Staubli VAL3: CMS_Module.pjx

--- CMS_Module.pjx ---
Parameters version=s8.10.2Cs9_BS1991 stackSize=20000 millimeterUnit=true
Program file=clkAirexOff.pgx
Program file=clkAirexOn.pgx
Program file=clkAllOff.pgx
Program file=clkAllOn.pgx
Program file=clkBack.pgx
Program file=clkCleanupChuck1.pgx
Program file=clkCleanupChuck2.pgx
Program file=clkDoAirex.pgx
Program file=clkDoModules.pgx
Program file=clkGlueGlass.pgx
Program file=clkPark1.pgx
Program file=clkPark2.pgx
Program file=clkValve0.pgx
Program file=clkValve1.pgx
Program file=clkValve10.pgx
Program file=clkValve11.pgx
Program file=clkValve12.pgx
Program file=clkValve13.pgx
Program file=clkValve14.pgx
Program file=clkValve15.pgx
Program file=clkValve16.pgx
Program file=clkValve17.pgx
Program file=clkValve2.pgx
Program file=clkValve3.pgx
Program file=clkValve4.pgx
Program file=clkValve5.pgx
Program file=clkValve6.pgx
Program file=clkValve7.pgx
Program file=clkValve8.pgx
Program file=clkValve9.pgx
Program file=clkValvePage.pgx
Program file=doAirex.pgx
Program file=doModules.pgx
Program file=glueGlass.pgx
Program file=goRemote.pgx
Program file=moveDown.pgx
Program file=moveStampUp.pgx
Program file=park1.pgx
Program file=print.pgx
Program file=selectedCheck.pgx
Program file=selectedClear.pgx
Program file=setSpeed.pgx
Program file=setValveStatus.pgx
Program file=socketServer.pgx
Program file=start.pgx
Program file=stop.pgx
Program file=toggleValve.pgx
Data file=CMS_Module.dtx

--- CMS_Module.dtx ---
bool bDoAirex = true
bool bGlueGlass
public dio doJ206_EtherCAT_Box_1__CPX_FB37__Q0 = {link=J206_EtherCAT\Box_1_(CPX-FB37)\%Q0}
public dio doJ206_EtherCAT_Box_1__CPX_FB37__Q1 = {link=J206_EtherCAT\Box_1_(CPX-FB37)\%Q1}
public dio doJ206_EtherCAT_Box_1__CPX_FB37__Q10 = {link=J206_EtherCAT\Box_1_(CPX-FB37)\%Q10}
public dio doJ206_EtherCAT_Box_1__CPX_FB37__Q11 = {link=J206_EtherCAT\Box_1_(CPX-FB37)\%Q11}
public dio doJ206_EtherCAT_Box_1__CPX_FB37__Q12 = {link=J206_EtherCAT\Box_1_(CPX-FB37)\%Q12}
public dio doJ206_EtherCAT_Box_1__CPX_FB37__Q13 = {link=J206_EtherCAT\Box_1_(CPX-FB37)\%Q13}
public dio doJ206_EtherCAT_Box_1__CPX_FB37__Q14 = {link=J206_EtherCAT\Box_1_(CPX-FB37)\%Q14}
public dio doJ206_EtherCAT_Box_1__CPX_FB37__Q15 = {link=J206_EtherCAT\Box_1_(CPX-FB37)\%Q15}
public dio doJ206_EtherCAT_Box_1__CPX_FB37__Q16 = {link=J206_EtherCAT\Box_1_(CPX-FB37)\%Q16}
public dio doJ206_EtherCAT_Box_1__CPX_FB37__Q17 = {link=J206_EtherCAT\Box_1_(CPX-FB37)\%Q17}
public dio doJ206_EtherCAT_Box_1__CPX_FB37__Q18 = {link=J206_EtherCAT\Box_1_(CPX-FB37)\%Q18}
public dio doJ206_EtherCAT_Box_1__CPX_FB37__Q19 = {link=J206_EtherCAT\Box_1_(CPX-FB37)\%Q19}
public dio doJ206_EtherCAT_Box_1__CPX_FB37__Q2 = {link=J206_EtherCAT\Box_1_(CPX-FB37)\%Q2}
public dio doJ206_EtherCAT_Box_1__CPX_FB37__Q20 = {link=J206_EtherCAT\Box_1_(CPX-FB37)\%Q20}
public dio doJ206_EtherCAT_Box_1__CPX_FB37__Q21 = {link=J206_EtherCAT\Box_1_(CPX-FB37)\%Q21}
public dio doJ206_EtherCAT_Box_1__CPX_FB37__Q22 = {link=J206_EtherCAT\Box_1_(CPX-FB37)\%Q22}
public dio doJ206_EtherCAT_Box_1__CPX_FB37__Q23 = {link=J206_EtherCAT\Box_1_(CPX-FB37)\%Q23}
public dio doJ206_EtherCAT_Box_1__CPX_FB37__Q24 = {link=J206_EtherCAT\Box_1_(CPX-FB37)\%Q24}
public dio doJ206_EtherCAT_Box_1__CPX_FB37__Q25 = {link=J206_EtherCAT\Box_1_(CPX-FB37)\%Q25}
public dio doJ206_EtherCAT_Box_1__CPX_FB37__Q26 = {link=J206_EtherCAT\Box_1_(CPX-FB37)\%Q26}
public dio doJ206_EtherCAT_Box_1__CPX_FB37__Q27 = {link=J206_EtherCAT\Box_1_(CPX-FB37)\%Q27}
public dio doJ206_EtherCAT_Box_1__CPX_FB37__Q28 = {link=J206_EtherCAT\Box_1_(CPX-FB37)\%Q28}
public dio doJ206_EtherCAT_Box_1__CPX_FB37__Q29 = {link=J206_EtherCAT\Box_1_(CPX-FB37)\%Q29}
public dio doJ206_EtherCAT_Box_1__CPX_FB37__Q3 = {link=J206_EtherCAT\Box_1_(CPX-FB37)\%Q3}
public dio doJ206_EtherCAT_Box_1__CPX_FB37__Q30 = {link=J206_EtherCAT\Box_1_(CPX-FB37)\%Q30}
public dio doJ206_EtherCAT_Box_1__CPX_FB37__Q31 = {link=J206_EtherCAT\Box_1_(CPX-FB37)\%Q31}
public dio doJ206_EtherCAT_Box_1__CPX_FB37__Q4 = {link=J206_EtherCAT\Box_1_(CPX-FB37)\%Q4}
public dio doJ206_EtherCAT_Box_1__CPX_FB37__Q5 = {link=J206_EtherCAT\Box_1_(CPX-FB37)\%Q5}
public dio doJ206_EtherCAT_Box_1__CPX_FB37__Q6 = {link=J206_EtherCAT\Box_1_(CPX-FB37)\%Q6}
public dio doJ206_EtherCAT_Box_1__CPX_FB37__Q7 = {link=J206_EtherCAT\Box_1_(CPX-FB37)\%Q7}
public dio doJ206_EtherCAT_Box_1__CPX_FB37__Q8 = {link=J206_EtherCAT\Box_1_(CPX-FB37)\%Q8}
public dio doJ206_EtherCAT_Box_1__CPX_FB37__Q9 = {link=J206_EtherCAT\Box_1_(CPX-FB37)\%Q9}
public dio switchMagnet = {link=FastIO\fOut0}
public dio switchVac0 = {link=ValveIO\valve1}
public dio switchVac1 = {link=ValveIO\valve2}
frame fPalette = {x=-254.28, y=175.62, z=30, rz=0.110016, fatherId=world[0]}
jointRs jInitialPosition = {j1=50, j2=50, j3=80, j4=15}
jointRs jRestPosition = {j1=70, j2=40, j3=80, j4=10}
mdesc mFast = {accel=20, vel=50, decel=20, leave=100}
mdesc mNomSpeed = {accel=10, vel=30, decel=10}
mdesc mSlow = {accel=5, vel=20, decel=5, tmax=99, rmax=99, leave=25, reach=25}
num airexValve[6]
  [0] = 12
  [1] = 6
  [3] = 13
  [4] = 7
  [5] = 1
num hdiValve[6]
  [0] = 14
  [1] = 8
  [2] = 2
  [3] = 16
  [4] = 10
  [5] = 4
num nError
num sensorValve[6]
  [0] = 15
  [1] = 9
  [2] = 3
  [3] = 17
  [4] = 11
  [5] = 5
num statusValves[32]
  [0] = 1
  [1] = 1
  [2] = 1
  [3] = 1
  [4] = 1
  [5] = 1
  [6] = 1
  [7] = 1
  [8] = 1
  [9] = 1
  [10] = 1
  [11] = 1
  [12] = 1
  [13] = 1
  [14] = 1
  [15] = 1
  [16] = 1
  [17] = 1
  [18] = 1
  [19] = 1
  [20] = 1
  [21] = 1
  [22] = 1
  [23] = 1
  [24] = 1
  [25] = 1
  [26] = 1
  [27] = 1
  [28] = 1
  [29] = 1
  [30] = 1
  [31] = 1
num waitGlue = 3
num waitShort = 1
pointRs airexFinal[6]
  [0] = {x=59, y=184, z=-97.69, rx=180, fatherId=fPalette[0]}
  [1] = {x=134, y=184, z=-97.69, rx=180, fatherId=fPalette[0]}
  [2] = {x=209, y=184, z=-97.69, rx=180, fatherId=fPalette[0]}
  [3] = {x=59, y=314, z=-97.69, rx=180, fatherId=fPalette[0]}
  [4] = {x=134, y=314, z=-97.69, rx=180, fatherId=fPalette[0]}
  [5] = {x=209, y=314, z=-97.69, rx=180, fatherId=fPalette[0]}
pointRs airexGlueStampEnd = {x=466.48, y=113.596594, z=-96.5, rx=180, ry=6.951996E-15, rz=0.0536958, fatherId=fPalette[0]}
pointRs airexGlueStampHome = {x=496, y=54, z=-97.69, rx=180, fatherId=fPalette[0]}
pointRs airexInitial[6]
  [0] = {x=59, y=113.6, z=-97.69, rx=180, fatherId=fPalette[0]}
  [1] = {x=134, y=113.6, z=-97.69, rx=180, fatherId=fPalette[0]}
  [2] = {x=209, y=113.6, z=-97.69, rx=180, fatherId=fPalette[0]}
  [3] = {x=59, y=144, z=-97.69, rx=180, fatherId=fPalette[0]}
  [4] = {x=134, y=144, z=-97.69, rx=180, fatherId=fPalette[0]}
  [5] = {x=209, y=144, z=-97.69, rx=180, fatherId=fPalette[0]}
pointRs chuck1[6]
  [0] = {x=59, y=39, z=-97.69, rx=180, fatherId=fPalette[0]}
  [1] = {x=134, y=39, z=-97.69, rx=180, fatherId=fPalette[0]}
  [2] = {x=209, y=39, z=-97.69, rx=180, fatherId=fPalette[0]}
  [3] = {x=59, y=79, z=-97.69, rx=180, fatherId=fPalette[0]}
  [4] = {x=134, y=79, z=-97.69, rx=180, fatherId=fPalette[0]}
  [5] = {x=209, y=79, z=-97.69, rx=180, fatherId=fPalette[0]}
pointRs chuck2[6]
  [0] = {x=291, y=54, z=-97.69, rx=180, fatherId=fPalette[0]}
  [1] = {x=361, y=54, z=-97.69, rx=180, fatherId=fPalette[0]}
  [2] = {x=291, y=119, z=-97.69, rx=180, fatherId=fPalette[0]}
  [3] = {x=361, y=119, z=-97.69, rx=180, fatherId=fPalette[0]}
  [4] = {x=291, y=184, z=-97.69, rx=180, fatherId=fPalette[0]}
  [5] = {x=361, y=184, z=-97.69, rx=180, fatherId=fPalette[0]}
pointRs gluePickPoint[6]
  [0] = {x=260, y=-15.8, z=-62.5, rx=180, ry=6.952208E-15, rz=0.0408868, fatherId=world[0]}
  [1] = {x=260, y=17.2, z=-62.5, rx=180, fatherId=world[0]}
  [2] = {x=290, y=-15.8, z=-62.5, rx=180, fatherId=world[0]}
  [3] = {x=290, y=17.2, z=-62.5, rx=180, fatherId=world[0]}
  [4] = {x=320, y=-15.8, z=-62.5, rx=180, fatherId=world[0]}
  [5] = {x=320, y=17.2, z=-62.5, rx=180, fatherId=world[0]}
pointRs hdiFinal[6]
  [0] = {x=59, y=249, z=-97.69, rx=180, fatherId=fPalette[0]}
  [1] = {x=134, y=249, z=-97.69, rx=180, fatherId=fPalette[0]}
  [2] = {x=209, y=249, z=-97.69, rx=180, fatherId=fPalette[0]}
  [3] = {x=59, y=379, z=-97.69, rx=180, fatherId=fPalette[0]}
  [4] = {x=134, y=379, z=-97.69, rx=180, fatherId=fPalette[0]}
  [5] = {x=209, y=379, z=-97.69, rx=180, fatherId=fPalette[0]}
pointRs pBasisRs = {x=-45.372705, y=215.0412411, z=72.706789, rx=180, ry=6.952541E-15, rz=0.0207374, fatherId=world[0]}
pointRs pFrameUrsprung = {x=-254.28, y=175.62, z=30, fatherId=world[0]}
pointRs pFrameX = {x=271.72, y=176.63, z=30, fatherId=world[0]}
pointRs pFrameY = {x=-255.12, y=613.62, z=30, fatherId=world[0]}
string colorOff = "beige"
string colorOn = "darkgreen"
string colorValveButton[32]
  [0] = "darkgreen"
  [1] = "darkgreen"
  [2] = "darkgreen"
  [3] = "darkgreen"
  [4] = "darkgreen"
  [5] = "darkgreen"
  [6] = "darkgreen"
  [7] = "darkgreen"
  [8] = "darkgreen"
  [9] = "darkgreen"
  [10] = "darkgreen"
  [11] = "darkgreen"
  [12] = "darkgreen"
  [13] = "darkgreen"
  [14] = "darkgreen"
  [15] = "darkgreen"
  [16] = "darkgreen"
  [17] = "darkgreen"
  [18] = "darkgreen"
  [19] = "darkgreen"
  [20] = "darkgreen"
  [21] = "darkgreen"
  [22] = "darkgreen"
  [23] = "darkgreen"
  [24] = "darkgreen"
  [25] = "darkgreen"
  [26] = "darkgreen"
  [27] = "darkgreen"
  [28] = "darkgreen"
  [29] = "darkgreen"
  [30] = "darkgreen"
  [31] = "darkgreen"
public tool tTool = {z=70, rz=-97.72, fatherId=flange[0]}
trsf trApproach = {z=-20}
trsf trStamp = {z=-6}
trsf trZsafe = {z=-70}
string colorVacuumStatus1
string statusDoAirex
string colorGray
string colorRunning
string colorCleanupChuck1
string statusCleanupChuck1
mdesc mVerySlow = {accel=2, vel=5, decel=2, tmax=5, rmax=5, leave=10, reach=10}
string statusDoModules
string statusCleanupChuck2
string colorCleanupChuck2
bool bDoModules
pointRs gluePickPoint2[6]
  [0] = {x=360, y=-25, z=-62.5, rx=180, ry=6.952208E-15, rz=0.0408868, fatherId=world[0]}
  [1] = {x=360, y=25, z=-62.5, rx=180, fatherId=world[0]}
  [2] = {x=410, y=-25, z=-62.5, rx=180, fatherId=world[0]}
  [3] = {x=410, y=25, z=-62.5, rx=180, fatherId=world[0]}
  [4] = {x=460, y=-25, z=-62.5, rx=180, fatherId=world[0]}
  [5] = {x=460, y=25, z=-62.5, rx=180, fatherId=world[0]}
pointRs moduleGlueStampHome = {x=436, y=54, z=-97.69, rx=180, ry=6.951996E-15, fatherId=fPalette[0]}
pointRs moduleGlueStampEnd = {x=466.48, y=156.596594, z=-96.5, rx=180, ry=6.951996E-15, rz=0.0536958, fatherId=fPalette[0]}
mdesc mExtremelySlow = {accel=0.05, vel=0.05, decel=0.05, tmax=0.04, rmax=0.04, leave=1, reach=1}
pointRs glueFirstPoint[2]
  [0] = {x=350, y=-15.8, z=-62.5, rx=180, ry=6.952208E-15, rz=0.0408868, fatherId=world[0]}
  [1] = {x=310, y=-25, z=-62.5, rx=180, rz=0.0408868, fatherId=world[0]}
trsf trZclose = {z=-10}
bool bSelectItem
bool bSelectedItems[6]
bool bSkipGlue
string colorError
string strStatus
trsf trZero
pointRs pSomewhere = {x=300, y=200, fatherId=world[0]}
trsf trPressTwo = {z=2}
trsf trUpTwo = {z=-8}
jointRs jPosition
string sPosition
bool bCleanup
num speedFactor
mdesc mSpeedArray[10]
  [0] = {accel=0.05, vel=0.05, decel=0.05, tmax=0.04, rmax=0.04, leave=1, reach=1}
  [1] = {accel=0.5, vel=0.5, decel=0.5, tmax=1, rmax=1, leave=2, reach=2}
  [2] = {accel=1, vel=1, decel=1, tmax=2, rmax=2, leave=2, reach=2}
  [3] = {accel=2, vel=2, decel=2, tmax=5, rmax=5, leave=5, reach=5}
  [4] = {accel=4, vel=5, decel=4, tmax=10, rmax=10, leave=10, reach=10}
  [5] = {accel=5, vel=7, decel=5, tmax=15, rmax=15, leave=20, reach=10}
  [6] = {accel=6, vel=10, decel=6, tmax=20, rmax=20, leave=20, reach=10}
  [7] = {accel=8, vel=15, decel=8, tmax=30, rmax=30, leave=40, reach=20}
  [8] = {accel=10, vel=20, decel=10, tmax=60, rmax=60, leave=40, reach=20}
  [9] = {accel=15, vel=30, decel=15, tmax=60, rmax=60, leave=80, reach=40}
trsf trDownTwo = {z=-2}
trsf trUpThree = {z=-9}
trsf trZverySafe = {z=-80}
string version
public sio sioSockets_server = {link=Socket\server}
string sReceiveMsg
string sSendMsg
public sio sioSockets_client = {link=Socket\client}
bool bGoRemote
string strTCPIP
bool bSockets
pointRs pGoRemoteTarget = {fatherId=fPalette[0]}

--- start.pgx ---
program start()
  local num nIndex
begin

  call print("Welcome to TEPX module production")
  version = "2024/12/20-07"

  strTCPIP = "TCP/IP sockets not activated"
  bSockets = false

  // -- required for local automatic?
  if esStatus() == 1
    setSafetyRestart()
  endIf
  if workingMode()==3
    if isPowered() == false
      enablePower()
    endIf
  endIf

  // -- define colors for valve buttons
  colorOff     = "beige"
  colorOn      = "darkgreen"
  colorGray    = "gray"
  colorRunning = "yellow"
  colorError   = "red"

  // -- initialize valve buttons and status
  call setValveStatus()
  for nIndex = 0 to 31
    if statusValves[nIndex] == 0
      colorValveButton[nIndex] = colorOff
    else
      colorValveButton[nIndex] = colorOn
    endIf
  endFor

  // -- initialize selection to be all on and bSelectItem to be off
  for nIndex = 0 to 5
    bSelectedItems[nIndex] = true
  endFor
  bSelectItem = false

  // -- initialize
  switchMagnet = false
  switchVac0   = false
  switchVac1   = false
  bDoAirex     = false
  bGlueGlass   = false
  bEndProgram  = false

  // -- airex valve indices
  airexValve[0]=12
  airexValve[1]=6
  airexValve[2]=0
  airexValve[3]=13
  airexValve[4]=7
  airexValve[5]=1

  // -- hdi valve indices
  hdiValve[0]=14
  hdiValve[1]=8
  hdiValve[2]=2
  hdiValve[3]=16
  hdiValve[4]=10
  hdiValve[5]=4

  // -- sensor valve indices
  sensorValve[0]=15
  sensorValve[1]=9
  sensorValve[2]=3
  sensorValve[3]=17
  sensorValve[4]=11
  sensorValve[5]=5

  colorVacuumStatus1 = colorOff
  colorCleanupChuck1 = colorOff
  colorCleanupChuck2 = colorOff

  statusDoAirex       = colorGray
  statusCleanupChuck1 = colorGray
  statusDoModules     = colorGray
  statusCleanupChuck2 = colorGray

  // -- define manual corrections for final placements
  // trXYCorrectionHDI = trXYZero
  trXYCorrectionHDI = trXYCorrection1

  // -- 4 is the production setting (mExtremelySlow = mSpeedArray[0])
  // -- all the rest have faster mExtremelySlow
  speedFactor = 4
  call setSpeed()

  // -- display user page
  userPage("firstpage")

  // -- this is here that fPalette is defined for manual jogs after program has started
  nError=setFrame(pFrameUrsprung, pFrameX, pFrameY, fPalette)
  resetMotion()
  movej(jInitialPosition, tTool, mNomSpeed)
  waitEndMove()

  taskCreate "doAirexTask", 10, doAirex()
  taskCreate "doModulesTask", 10, doModules()
  taskCreate "doGlueGlass", 10, glueGlass()

  // Note: This is activated only after enabling arm power or move/hold button?!
  taskCreate "socketServerTask", 10, socketServer()


  while true
    jPosition = herej()
    sPosition = toString("6.3", jPosition.j3)
    sMovementID = toString("6.3", getMoveId())
  endWhile

end

--- clkCleanupChuck1.pgx ---
program clkCleanupChuck1()
  local num nAirexIdx
begin
  switchMagnet=false
  statusCleanupChuck1 = colorRunning

  call selectedCheck()
  call print("cleanup (airex) start")

  // -- pick vacuum chuck1's and put them back to their original place
  for nAirexIdx=0 to 5
    if !bSelectItem or (bSelectedItems[nAirexIdx]==true)
      call print("put away chuck " + toString("1.0", nAirexIdx))
      // -- move over final airex position (where the chuck is from gluing) and down
      // -- for edge positions make a curve to avoid hitting side bar
      if nAirexIdx == 0 or nAirexIdx == 3
        movej(appro(airexInitial[1], trZsafe), tTool, mFast)
      endIf

      call moveDown(airexFinal[nAirexIdx], mSlow, trZero, false)

      // -- lift chuck1
      switchMagnet=true
      delay(waitShort)
      movel(appro(airexFinal[nAirexIdx], trZsafe), tTool, mSlow)
      //waitEndMove()

      // -- move over/to initial chuck position
      // -- for edge positions make a curve to avoid hitting side bar
      if nAirexIdx == 0 or nAirexIdx == 3
        movej(appro(airexInitial[1], trZsafe), tTool, mFast)
      endIf
      call moveDown(chuck1[nAirexIdx], mSlow, trZero, false)

      // -- release it
      switchMagnet=false

      // -- move up
      movel(appro(chuck1[nAirexIdx], trZsafe), tTool, mSlow)
    endIf
  endFor

  // -- move back somewhere
  call print("parking robot")
  waitEndMove()
  movej(jInitialPosition, tTool, mFast)
  waitEndMove()
  statusCleanupChuck1 = colorOn
  statusDoAirex = colorGray
  call print("cleanup (airex) done")
  //call selectedClear()

end

--- clkCleanupChuck2.pgx ---
program clkCleanupChuck2()
  local num nIdx
begin
  switchMagnet=false
  statusCleanupChuck2 = colorRunning

  call selectedCheck()
  call print("cleanup (modules) start")

  // -- pick vacuum chuck2's and put them back to their original place
  for nIdx=0 to 5
    if !bSelectItem or (bSelectedItems[nIdx]==true)
      call print("put away chuck " + toString("1.0", nIdx))
      // -- move over final hdi position (where the chuck is from gluing) and down
      // -- for edge positions make a curve to avoid hitting side bar
      if nIdx == 0 or nIdx == 3
        movej(appro(airexInitial[1], trZsafe), tTool, mFast)
      endIf

      // test
      if(nIdx==3)
        trXYCorrectionHDI = trXYZero
      else
        trXYCorrectionHDI = trXYCorrection1
      endIf

      call moveDown(hdiFinal[nIdx], mSlow, trPressTwo, false, trXYCorrectionHDI)

      // -- lift chuck2
      switchMagnet=true
      delay(waitShort)
      movel(appro(hdiFinal[nIdx], trZsafe), tTool, mSlow)
      //waitEndMove()

      // -- move over/to initial chuck position
      // -- for edge positions make a curve to avoid hitting side bar
      if nIdx == 0 or nIdx == 3
        movej(appro(airexInitial[1], trZsafe), tTool, mFast)
      endIf
      call moveDown(chuck2[nIdx], mSlow, trZero, false, trXYZero)

      // -- release it
      switchMagnet=false

      // -- move up
      movel(appro(chuck2[nIdx], trZsafe), tTool, mSlow)
    endIf
  endFor

  // -- move back somewhere
  call print("parking robot")
  waitEndMove()
  movej(jInitialPosition, tTool, mFast)
  waitEndMove()
  call print("cleanup (modules) done")
  statusCleanupChuck2 = colorOn
  statusDoModules = colorGray
  //call selectedClear()

end

--- clkDoTest.pgx ---
program clkDoTest()
begin
  bDoTest=true
end

--- clkPark2.pgx ---
program clkPark2()
begin
  // -- move back to initial position
  resetMotion()
  movej(jInitialPosition,tTool,mNomSpeed)
  waitEndMove()
end

--- clkStop.pgx ---
program clkStop()
begin
  bDoAirex = false
  bDoModules = false
  bCleanup = false
end

--- doAirex.pgx ---
program doAirex()
  local num nAirexIdx
  local bool vacuumCheckDone
begin
  vacuumCheckDone = false
  while true
    call parkEndProgram()

    if bDoAirex==true
      call selectedCheck()
      call print("starting doAirex")
      statusDoAirex = colorRunning

      // -- check that relevant vacuum is active
      if !bSelectItem
        // -- check all
        call print("check vacuum on all")
        delay(waitShort)
        for nAirexIdx = 0 to 5
          // -- check only the sensor valves, not the AIREX frame valves (don't care about those)
          if statusValves[sensorValve[nAirexIdx]] == 0
            bDoAirex = false
            statusDoAirex = colorError
            call print("Error: no vacuum at position " + toString("1.0", nAirexIdx))
          endIf
        endFor
      else
        // -- check only those that are selected
        call print("check vacuum on selection")
        delay(waitShort)
        for nAirexIdx = 0 to 5
          if statusValves[sensorValve[nAirexIdx]] == 0 and (bSelectedItems[nAirexIdx]==true)
            bDoAirex = false
            statusDoAirex = colorError
            call print("Error: no vacuum at position " + toString("1.0", nAirexIdx))
          endIf
        endFor
      endIf
      vacuumCheckDone = true
      if bDoAirex == false
        call print("Fix missing vacuum and try again")
        vacuumCheckDone = false
      endIf

    endIf

    // -- return above does not work. It terminates the task!
    if bDoAirex==true and vacuumCheckDone==true
      call setSpeed()

      if bSkipGlue[0]==false
        call print("picking glue stamp")
        // -- pick glue stamp
        call moveDown(airexGlueStampHome, mSlow, trZero, false, trXYZero)
        waitEndMove()
        movel(appro(airexGlueStampHome, trPressTwo), tTool, mVerySlow)
        waitEndMove()
        delay(waitShort)
        switchMagnet=true
        movel(appro(airexGlueStampHome, trZsafe), tTool, mSlow)

        call parkEndProgram()

        // -- double-dip stamp into glue before starting the normal procedure
        call moveDown(glueFirstPoint[1], mSlow, trZero, false, trXYZero)
        delay(waitGlue)
        call moveStampUp(glueFirstPoint[1], mVerySlow, trXYZero)
        call moveDown(glueFirstPoint[0], mSlow, trZero, false, trXYZero)
        delay(waitGlue)
        call moveStampUp(glueFirstPoint[0], mVerySlow, trXYZero)

        call parkEndProgram()

        // -- apply glue stamp to all positions:
        //    divide approach onto /from glue position into two steps
        //    (1) slowly to trApproach above it
        //    (2) extremely slowly down to/up from glue to trApproach
        for nAirexIdx=0 to 5
          if !bSelectItem or (bSelectedItems[nAirexIdx]==true)
            call setSpeed()
            if bDoAirex==true

              call parkEndProgram()

              call print("getting glue for position " + toString("1.0", nAirexIdx))
              call moveDown(gluePickPoint[nAirexIdx], mSlow, trZero, false, trXYZero)
              delay(waitGlue)

              call moveStampUp(gluePickPoint[nAirexIdx], mVerySlow, trXYZero)

              call parkEndProgram()

              // -- move to where the glue should be applied (the final airex position)
              call print("applying glue to position " + toString("1.0", nAirexIdx))
              call moveDown(airexFinal[nAirexIdx], mSlow, trStamp, false, trXYZero)
              delay(waitGlue)
              call moveStampUp(airexFinal[nAirexIdx], mVerySlow, trXYZero)
            endIf
          endIf
        endFor

        // -- Drop glue stamp
        call setSpeed()
        call print("put away glue stamp")
        call moveDown(airexGlueStampEnd, mSlow, trPressTwo, false, trXYZero)
        waitEndMove()
        switchMagnet = false
        movel(appro(airexGlueStampEnd, trZsafe), tTool, mNomSpeed)
      endIf

      if !bSelectItem
        call print("handling all airex frames")
      else
        call print("handling selected airex frames")
      endIf

      // -- pick weighted vacuum chucks and lift airex frames to HDIs
      for nAirexIdx=0 to 5
        if !bSelectItem or (bSelectedItems[nAirexIdx]==true)
          call setSpeed()
          if bDoAirex==true
            // -- move over/to chuck
            call moveDown(chuck1[nAirexIdx], mSlow, trZero, false, trXYZero)
            // -- the following cures the click when the chuck 'jumps' up a bit
            waitEndMove()
            movel(appro(chuck1[nAirexIdx], trPressTwo), tTool, mVerySlow)
            waitEndMove()

            // -- pick chuck and move up
            switchMagnet=true
            delay(waitShort)
            call print("picking airex frame " + toString("1.0", nAirexIdx))
            movel(appro(chuck1[nAirexIdx], trZsafe), tTool, mSlow)

            // -- move with chuck to airex position
            call moveDown(airexInitial[nAirexIdx], mSlow, trZero, false, trXYZero)

            // -- release airex vacuum to allow picking up
            if statusValves[airexValve[nAirexIdx]]==1
              call toggleValve(airexValve[nAirexIdx])
            endIf
            delay(waitShort)
            switchVac0=true
            switchVac1=true
            delay(waitShort)

            // -- move up with airex frame
            call print("placing airex frame " + toString("1.0", nAirexIdx))
            movel(appro(airexInitial[nAirexIdx], trZclose), tTool, mSlow)
            movel(appro(airexInitial[nAirexIdx], trZsafe), tTool, mNomSpeed)

            call parkEndProgram()

            // -- move to final airex position and put down
            call moveDown(airexFinal[nAirexIdx], mVerySlow, trZero, false, trXYZero)
            switchVac0   = false
            switchVac1   = false
            switchMagnet = false

            delay(waitShort)

            // -- move up again
            movel(appro(airexFinal[nAirexIdx], trZclose), tTool, mSlow)
            movel(appro(airexFinal[nAirexIdx], trZsafe), tTool, mNomSpeed)
          endIf
        endIf
      endFor

      // -- move back somewhere
      call print("parking robot")
      //waitEndMove()
      movej(jInitialPosition, tTool, mFast)
      waitEndMove()
      statusDoAirex = colorOn

      //call selectedClear()
      bDoAirex=false
      call print("glue airex done")
    endIf
  endWhile

end

--- doModules.pgx ---
program doModules()
  local num nIdx
  local bool vacuumCheckDone
begin
  vacuumCheckDone = false
  while true
    if bDoModules==true
      call selectedCheck()
      call print("starting doModules")
      statusDoModules = colorRunning
      statusCleanupChuck1 = colorGray

      // -- check that relevant vacuum is active
      if !bSelectItem
        // -- check all
        call print("check vacuum on all")
        delay(waitShort)
        for nIdx = 0 to 5
          if statusValves[sensorValve[nIdx]] == 0
            bDoModules = false
            statusDoModules = colorError
            call print("Error: no vacuum at position" + toString("1.0", nIdx))
          endIf
        endFor
      else
        // -- check only those that are selected
        call print("check vacuum on selection")
        delay(waitShort)
        for nIdx = 0 to 5
          if statusValves[sensorValve[nIdx]] == 0 and bSelectedItems[nIdx] == true
            bDoModules = false
            statusDoModules = colorError
            call print("Error: no vacuum at position" + toString("1.0", nIdx))
          endIf
        endFor
      endIf
      vacuumCheckDone = true
      if bDoModules == false
        call print("Fix missing vacuum and try again")
        vacuumCheckDone = false
      endIf
    endIf

    // -- return above does not work. It terminates the task!
    if bDoModules==true and vacuumCheckDone==true
      statusDoModules = colorRunning
      call setSpeed()

      if bSkipGlue[0] == false
        call print("picking glue stamp")
        // -- pick glue stamp
        call moveDown(moduleGlueStampHome, mFast, trZero, false, trXYZero)
        waitEndMove()
        movel(appro(moduleGlueStampHome, trPressTwo), tTool, mVerySlow)
        waitEndMove()
        delay(waitShort)
        switchMagnet=true
        movel(appro(moduleGlueStampHome, trZsafe), tTool, mSlow)

        call parkEndProgram()

        // -- double-dip stamp into glue before starting the normal procedure
        call print("pre-dip glue stamp")
        call moveDown(glueFirstPoint[1], mFast, trOne, false, trXYZero)
        waitEndMove()
        delay(waitGlue)
        call moveStampUp(glueFirstPoint[1], mSlow, trXYZero)

        call moveDown(glueFirstPoint[0], mSlow, trOne, false, trXYZero)
        waitEndMove()
        delay(waitGlue)
        call moveStampUp(glueFirstPoint[0], mSlow, trXYZero)

        call parkEndProgram()

        // -- apply glue stamp to all positions
        //    divide approach onto /from glue position into two steps
        //    (1) slowly to trApproach above it
        //    (2) extremely slowly up from glue to trApproach
        for nIdx=0 to 5
          if !bSelectItem or (bSelectedItems[nIdx]==true)
            call setSpeed()
            if bDoModules==true
              call print("getting glue for position " + toString("1.0", nIdx))
              call moveDown(gluePickPoint2[nIdx], mSlow, trOne, false, trXYZero)
              waitEndMove()
              delay(waitGlue)

              call moveStampUp(gluePickPoint2[nIdx], mSlow, trXYZero)

              call parkEndProgram()

              // -- move to where the glue should be applied (the final hdi position)
              call print("applying glue to position " + toString("1.0", nIdx))
              call moveDown(hdiFinal[nIdx], mVerySlow, trStamp, false, trXYZero)
              //call moveDown(hdiFinal[nIdx], mVerySlow, trStamp, false, trXYstampOffset)
              waitEndMove()
              delay(waitGlue)
              call moveStampUp(hdiFinal[nIdx], mExtremelySlow, trXYZero)
              //call moveStampUp(hdiFinal[nIdx], mExtremelySlow, trXYstampOffset)
            endIf
          endIf
        endFor

        // -- Drop glue stamp
        call setSpeed()
        call print("put away glue stamp")
        call moveDown(moduleGlueStampEnd, mFast, trPressTwo, false, trXYZero)
        waitEndMove()
        switchMagnet = false
        movel(appro(moduleGlueStampEnd, trZsafe), tTool, mNomSpeed)
      endIf

      if !bSelectItem
        call print("handling all modules")
      else
        call print("handling selected modules")
      endIf

      // -- pick weighted vacuum chucks and lift airex frames to HDIs
      for nIdx=0 to 5
        if !bSelectItem or (bSelectedItems[nIdx]==true)
          call setSpeed()
          if bDoModules==true
            // -- move over/to chuck
            call moveDown(chuck2[nIdx], mSlow, trZero, false, trXYZero)
            // -- the following cures the click when the chuck 'jumps' up a bit
            waitEndMove()
            movel(appro(chuck2[nIdx], trPressTwo), tTool, mVerySlow)
            waitEndMove()

            // -- pick it
            switchMagnet = true
            delay(waitShort)
            call print("picking module " + toString("1.0", nIdx))
            movel(appro(chuck2[nIdx], trZsafe), tTool, mSlow)

            // -- move to hdi initial location (where the airex frame had been glued) and lower
            call moveDown(airexFinal[nIdx], mSlow, trZero, false, trXYZero)

            // -- release hdi vacuum to allow picking up
            call toggleValve(hdiValve[nIdx])
            delay(waitShort)
            switchVac0=true
            switchVac1=true
            delay(waitShort)

            // -- move up
            call print("placing hdi " + toString("1.0", nIdx))
            movel(appro(airexFinal[nIdx], trZclose), tTool, mSlow)
            movel(appro(airexFinal[nIdx], trZsafe), tTool, mNomSpeed)

            // -- move to final location
            call moveDown(hdiFinal[nIdx], mVerySlow, trZero, false, trXYCorrectionHDI)
            switchVac0   = false
            switchVac1   = false
            switchMagnet = false

            delay(waitShort)

            // -- move up again
            movel(appro(hdiFinal[nIdx], trZclose), tTool, mSlow)
            movel(appro(hdiFinal[nIdx], trZsafe), tTool, mNomSpeed)
          endIf

        endIf
      endFor

      // -- move back somewhere
      call print("parking robot")
      movej(jInitialPosition, tTool, mFast)
      waitEndMove()
      statusDoModules = colorOn

      //call selectedClear()
      bDoModules = false
      call print("glue modules done")
    endIf
  endWhile

end

--- doTest.pgx ---
program doTest()
begin
  call park1()

  while true

    if bDoTest==true
      if statusValves[hdiValve[0]]==0 or statusValves[sensorValve[0]]==0
        userPageAlert("No vaccum applied to airex #0. Fix this first!")
        return
      elseIf statusValves[hdiValve[1]]==0
        userPageAlert("No vaccum applied to airex #1. Fix this first!")
        return
      elseIf statusValves[hdiValve[2]]==0
        userPageAlert("No vaccum applied to airex #2. Fix this first!")
        return
      elseIf statusValves[hdiValve[3]]==0
        userPageAlert("No vaccum applied to airex #3. Fix this first!")
        return
      elseIf statusValves[hdiValve[4]]==0
        userPageAlert("No vaccum applied to airex #4. Fix this first!")
        return
      elseIf statusValves[hdiValve[5]]==0
        userPageAlert("No vaccum applied to airex #5. Fix this first!")
        return
      endIf
    endIf

  endWhile
end

--- glueGlass.pgx ---
program glueGlass()
  local num nIdx
begin
  while true
    delay(1)
    if bGlueGlass==true
      call selectedCheck()
      call print("starting glueGlass test")

      // -- check that relevant vacuum is active
      if !bSelectItem
        // -- check all
        call print("check vacuum on all")
        delay(waitShort)
        for nIdx = 0 to 5
          if statusValves[hdiValve[nIdx]] == 0
            bGlueGlass = false
            call print("Error: no HDI vacuum at position " + toString("1.0", nIdx))
          endIf
          if statusValves[sensorValve[nIdx]] == 0
            bGlueGlass = false
            call print("Error: no sensor vacuum at position " + toString("1.0", nIdx))
          endIf
        endFor
      else
        // -- check only those that are selected
        call print("check vacuum on selection")
        delay(waitShort)
        for nIdx = 0 to 5
          if statusValves[hdiValve[nIdx]] == 0 and (bSelectedItems[nIdx]==true)
            bGlueGlass = false
            call print("Error: no HDI vacuum at position " + toString("1.0", nIdx))
          endIf
          if statusValves[sensorValve[nIdx]] == 0 and (bSelectedItems[nIdx]==true)
            bGlueGlass = false
            call print("Error: no sensor vacuum at position " + toString("1.0", nIdx))
          endIf
        endFor
      endIf
      if bGlueGlass == false
        call print("Fix missing vacuum and try again")
      endIf

    endIf

    // -- return above does not work. It terminates the task!
    if bGlueGlass==true
      call setSpeed()

      if bSkipGlue[0]==false
        call print("picking module glue stamp")
        // -- pick glue stamp
        call moveDown(moduleGlueStampHome, mFast, trZero, false, trXYZero)
        waitEndMove()
        movel(appro(moduleGlueStampHome, trPressTwo), tTool, mVerySlow)
        waitEndMove()
        delay(waitShort)
        switchMagnet=true
        movel(appro(moduleGlueStampHome, trZsafe), tTool, mSlow)

        call parkEndProgram()

        // -- double-dip stamp into glue before starting the normal procedure
        call print("pre-dip glue stamp")
        call moveDown(glueFirstPoint[1], mFast, trOne, false, trXYZero)
        waitEndMove()
        delay(waitGlue)
        call moveStampUp(glueFirstPoint[1], mSlow, trXYZero)

        call moveDown(glueFirstPoint[0], mSlow, trOne, false, trXYZero)
        waitEndMove()
        delay(waitGlue)
        call moveStampUp(glueFirstPoint[0], mSlow, trXYZero)

        call parkEndProgram()

        // -- apply glue stamp to all positions:
        //    divide approach onto/from glue position into two steps
        //    (1) slowly to trApproach above it
        //    (2) extremely slowly up from glue to trApproach
        for nIdx=0 to 5
          if !bSelectItem or (bSelectedItems[nIdx]==true)
            call setSpeed()
            if bGlueGlass==true
              call print("getting glue for position " + toString("1.0", nIdx))
              call moveDown(gluePickPoint2[nIdx], mSlow, trOne, false, trXYZero)
              waitEndMove()
              delay(waitGlue)

              call moveStampUp(gluePickPoint2[nIdx], mSlow, trXYZero)

              call parkEndProgram()

              // -- move to where the glue should be applied (the final hdi position)
              call print("applying glue to position " + toString("1.0", nIdx))
              call moveDown(hdiFinal[nIdx], mVerySlow, trStamp, false, trXYZero)
              //call moveDown(hdiFinal[nIdx], mVerySlow, trStamp, false, trXYstampOffset)
              waitEndMove()
              delay(waitGlue)
              call moveStampUp(hdiFinal[nIdx], mExtremelySlow, trXYZero)
              //call moveStampUp(hdiFinal[nIdx], mExtremelySlow, trXYstampOffset)
            endIf
          endIf
        endFor

        // -- Drop glue stamp
        call setSpeed()
        call print("put away glue stamp")
        call moveDown(moduleGlueStampEnd, mSlow, trPressTwo, false, trXYZero)
        waitEndMove()
        switchMagnet = false
        movel(appro(moduleGlueStampEnd, trZsafe), tTool, mNomSpeed)
      endIf

      if !bSelectItem
        call print("handling all glasses")
      else
        call print("handling selected glasses")
      endIf

      // -- pick weighted vacuum chucks and lift glasses to final locations
      for nIdx=0 to 5
        if !bSelectItem or (bSelectedItems[nIdx]==true)
          call setSpeed()
          if bGlueGlass==true
            // -- move over/to chuck
            call moveDown(chuck2[nIdx], mSlow, trZero, false, trXYZero)
            // -- the following cures the click when the chuck 'jumps' up a bit
            waitEndMove()
            movel(appro(chuck2[nIdx], trPressTwo), tTool, mVerySlow)
            waitEndMove()

            call parkEndProgram()

            // -- pick chuck and move up
            switchMagnet=true
            delay(waitShort)
            call print("picking module frame " + toString("1.0", nIdx))
            movel(appro(chuck2[nIdx], trZsafe), tTool, mSlow)

            call parkEndProgram()

            // -- move with chuck to hdi glass(!) position
            call moveDown(glassInitial[nIdx], mSlow, trZero, true, trXYZero)

            // -- release hdi vacuum to allow picking up hdi glass
            if statusValves[hdiValve[nIdx]]==1
              call toggleValve(hdiValve[nIdx])
            endIf
            delay(waitShort)
            switchVac0=true
            switchVac1=true
            delay(waitShort)

            // -- move up with hdi glass
            call print("placing hdi glass " + toString("1.0", nIdx))
            movel(appro(glassInitial[nIdx], trZclose), tTool, mSlow)
            movel(appro(glassInitial[nIdx], trZsafe), tTool, mNomSpeed)

            call parkEndProgram()

            // -- move to final HDI position and put down
            call moveDown(hdiFinal[nIdx], mVerySlow, trZero, true, trXYZero)
            switchVac0   = false
            switchVac1   = false
            switchMagnet = false

            delay(waitShort)

            // -- move up again
            movel(appro(hdiFinal[nIdx], trZclose), tTool, mSlow)
            movel(appro(hdiFinal[nIdx], trZsafe), tTool, mNomSpeed)

            call parkEndProgram()
          endIf
        endIf
      endFor

      // -- move back somewhere
      call print("parking robot")
      //waitEndMove()
      movej(jInitialPosition, tTool, mFast)
      waitEndMove()

      //call selectedClear()
      bGlueGlass=false
      call print("glueGlass done")
    endIf
  endWhile

end

--- goRemote.pgx ---
program goRemote()
begin
  call setSpeed()
  movel(pGoRemoteTarget, tTool, mNomSpeed)
  waitEndMove()
end

--- moveDown.pgx ---
program moveDown(pointRs where, mdesc finalSpeed, trsf finalAppro, bool meticulous, trsf xyTrsf)
  local mdesc speed[3]
begin
  // Note: finalSpeed is not taken literally!
  if finalSpeed == mVerySlow
    speed[0] = mFast
    speed[1] = mSlow
    speed[2] = mVerySlow
  elseIf finalSpeed == mSlow
    speed[0] = mFast
    speed[1] = mSlow
    speed[2] = mSlow
  else
    speed[0] = mFast
    speed[1] = mFast
    speed[2] = mSlow
  endIf

  //movej(appro(where, trZsafe*xyTrsf), tTool, speed[0])
  movej(appro(where, trZsafe), tTool, speed[0])
  if meticulous
    waitEndMove()
  endIf

  // -- move down with decreasing speeds. Not sure whether this gets "blended" away
  //movej(appro(where, trZclose*xyTrsf), tTool, speed[1])
  //movej(appro(where, finalAppro*xyTrsf), tTool, speed[2])

  movej(appro(where, trZclose), tTool, speed[1])
  movej(appro(where, finalAppro), tTool, speed[2])
  waitEndMove()
end

--- moveStampUp.pgx ---
program moveStampUp(pointRs where, mdesc iniSpeed, trsf xyTrsf)
begin
  movej(appro(where, trUpThree*xyTrsf), tTool, iniSpeed)
  if iniSpeed == mExtremelySlow
    waitEndMove()
  endIf

  if iniSpeed == mExtremelySlow
    movej(appro(where, trZclose*xyTrsf), tTool, mVerySlow)
    waitEndMove()
  else
    movej(appro(where, trZclose*xyTrsf), tTool, mSlow)
  endIf

  movej(appro(where, trZsafe*xyTrsf), tTool, mSlow)
end

--- park1.pgx ---
program park1()
begin
  // -- move back to rest position
  resetMotion()
  movej(jRestPosition,tTool,mNomSpeed)
  waitEndMove()
end

--- parkEndProgram.pgx ---
program parkEndProgram()
  local jointRs jPos
begin
  if bEndProgram==true
    call print("end program, put robot into safe state")

    statusDoAirex       = colorError
    statusCleanupChuck1 = colorError
    statusCleanupChuck2 = colorError
    statusDoModules     = colorError

    jPos = herej()
    call print("end program: stopMove at here.z = "  + toString("6.3", jPos.j3))
    delay(1)
    stopMove()

   // jPos = herej()
    call print("end program: resetMotion at here.z = "  + toString("6.3", jPos.j3))
    delay(1)
    resetMotion()


    // -- move up to safe z position from wherever you are
    jPos.j3 = 70
    call print("end program: move up")
    movej(jPos, tTool, mSlow)
    waitEndMove()

    // -- move over end of foil, deposit anything connected
    call print("end program: move to appro(parkEndPoint, trZsafe)")
    movej(appro(parkEndPoint, trZsafe), tTool, mNomSpeed)
    waitEndMove()
    call print("end program: move to appro(parkEndPoint, trZero)")
    movej(appro(parkEndPoint, trZero), tTool, mSlow)
    waitEndMove()
    call print("end program: drop tool")
    switchMagnet = false
    switchVac0   = false
    switchVac1   = false
    delay(1)

    // -- move up
    call print("end program: move up")
    movej(appro(parkEndPoint, trZsafe), tTool, mNomSpeed)
    waitEndMove()

    // -- move to normal rest position
    call print("end program: move to normal rest position")
    movej(jInitialPosition, tTool, mFast)
    waitEndMove()
    resetMotion()

    //taskKill("doAirexTask")
    //taskKill("doModulesTask")
    //taskKill("doGlueGlass")

    bEndProgram = false
    disablePower()
    call print("program ended, now what?")
  endIf

end

--- selectedCheck.pgx ---
program selectedCheck()
begin
   if bSelectedItems[0]==true and bSelectedItems[1]==true and bSelectedItems[2]==true and bSelectedItems[3]==true and bSelectedItems[4]==true and bSelectedItems[5]==true
    bSelectItem = false
  else
    bSelectItem = true
  endIf

end

--- selectedClear.pgx ---
program selectedClear()
begin
  if bSelectItem
    bSelectedItems[0] = true
    bSelectedItems[1] = true
    bSelectedItems[2] = true
    bSelectedItems[3] = true
    bSelectedItems[4] = true
    bSelectedItems[5] = true
  endIf
  bSelectItem = false
end

--- setSpeed.pgx ---
program setSpeed()
begin
  if speedFactor <= 1
    mExtremelySlow = mSpeedArray[1]
    mVerySlow      = mSpeedArray[1]
    mSlow          = mSpeedArray[2]
    mNomSpeed      = mSpeedArray[4]
    mFast          = mSpeedArray[5]
  elseIf speedFactor == 2
    mExtremelySlow = mSpeedArray[2]
    mVerySlow      = mSpeedArray[2]
    mSlow          = mSpeedArray[3]
    mNomSpeed      = mSpeedArray[5]
    mFast          = mSpeedArray[7]
   elseIf speedFactor == 3
    mExtremelySlow = mSpeedArray[3]
    mVerySlow      = mSpeedArray[3]
    mSlow          = mSpeedArray[4]
    mNomSpeed      = mSpeedArray[6]
    mFast          = mSpeedArray[8]
  elseIf speedFactor == 4
    mExtremelySlow = mSpeedArray[0]
    mVerySlow      = mSpeedArray[4]
    mSlow          = mSpeedArray[5]
    mNomSpeed      = mSpeedArray[7]
    mFast          = mSpeedArray[9]
  elseIf speedFactor >= 5
    mExtremelySlow = mSpeedArray[3]
    mVerySlow      = mSpeedArray[4]
    mSlow          = mSpeedArray[5]
    mNomSpeed      = mSpeedArray[7]
    mFast          = mSpeedArray[9]
endIf

end

--- socketServer.pgx ---
program socketServer()
  local num i
  local bool l_bError
  local num l_nResult
  local num l_nReceiveByte
  local num numSendMsg[255]
begin
  clearBuffer(sioSockets_server)
  strTCPIP = "TCP/IP sockets server is ready"
  delay(0)

  while true

    sReceiveMsg=""

    if bSockets
      do
        l_nResult = sioGet(sioSockets_server, l_nReceiveByte)
        sReceiveMsg = sReceiveMsg + chr(l_nReceiveByte)

        // Note: 10 = LF
        //       13 = CR // this is set as "End of string"
        // Linux  - Lines end with only a <LF> character
        // Macintosh (Mac OSX) - Lines end with only a <LF> character
        // NOTE: tcpip.swift sends a 13?!?!
      until l_nResult!=1 or l_nReceiveByte==13

      //call print("receive ->" + sReceiveMsg + "<-")
      strTCPIP = sReceiveMsg
      delay(0.5)

      if find(strTCPIP, "goRemote") == 0
        //        pGoRemote[0] = {134,	249,	-90.69, 0., 0., 0.}
        pGoRemoteTarget[0].trsf.x = 130
        pGoRemoteTarget[0].trsf.y = 150
        pGoRemoteTarget[0].trsf.z = -80
        pGoRemoteTarget[0].trsf.rx = 180.0
        call goRemote()
      endIf


      //    sSendMsg = "ss received ->" + sReceiveMsg + "<-"
      //    for i = 0 to len(sSendMsg)
      //      numSendMsg[i] = asc(sSendMsg[i],0)
      //    endFor
      //    sioSet(sioSockets_server, numSendMsg)

      //sioSet()
      //    // write
      //    ? sSendMsg = "Hello I'm the cms-ts2-60 server "
      //    for i = 0 to len(sSendMsg)-1
      //      l_nResult=sioSet(sioSockets_server, asc(sSendMsg,i))
      //      if l_nResult != 1
      //        i = len(sSendMsg)
      //        l_bError = true
      //      endIf
      //    endFor
      //    // connection will close
      //    ? "TCP/IP server end"
      //    wait(false)
    endIf
  endWhile
end

--- toggleValve.pgx ---
program toggleValve(num iValve)
begin
  if statusValves[iValve]==1
    statusValves[iValve]=0
    colorValveButton[iValve]=colorOff
    switch iValve
      case 0
        doJ206_EtherCAT_Box_1__CPX_FB37__Q0[0]=false
      break
      case 1
        doJ206_EtherCAT_Box_1__CPX_FB37__Q1[0]=false
      break
      case 2
        doJ206_EtherCAT_Box_1__CPX_FB37__Q2[0]=false
      break
      case 3
        doJ206_EtherCAT_Box_1__CPX_FB37__Q3[0]=false
      break
      case 4
        doJ206_EtherCAT_Box_1__CPX_FB37__Q4[0]=false
      break
      case 5
        doJ206_EtherCAT_Box_1__CPX_FB37__Q5[0]=false
      break
      case 6
        doJ206_EtherCAT_Box_1__CPX_FB37__Q6[0]=false
      break
      case 7
        doJ206_EtherCAT_Box_1__CPX_FB37__Q7[0]=false
      break
      case 8
        doJ206_EtherCAT_Box_1__CPX_FB37__Q8[0]=false
      break
      case 9
        doJ206_EtherCAT_Box_1__CPX_FB37__Q9[0]=false
      break
      case 10
        doJ206_EtherCAT_Box_1__CPX_FB37__Q10[0]=false
      break
      case 11
        doJ206_EtherCAT_Box_1__CPX_FB37__Q11[0]=false
      break
      case 12
        doJ206_EtherCAT_Box_1__CPX_FB37__Q12[0]=false
      break
      case 13
        doJ206_EtherCAT_Box_1__CPX_FB37__Q13[0]=false
      break
      case 14
        doJ206_EtherCAT_Box_1__CPX_FB37__Q14[0]=false
      break
      case 15
        doJ206_EtherCAT_Box_1__CPX_FB37__Q15[0]=false
      break
      case 16
        doJ206_EtherCAT_Box_1__CPX_FB37__Q16[0]=false
      break
      case 17
        doJ206_EtherCAT_Box_1__CPX_FB37__Q17[0]=false
      break
    endSwitch
  else
    statusValves[iValve]=1
    colorValveButton[iValve]=colorOn
    switch iValve
      case 0
        doJ206_EtherCAT_Box_1__CPX_FB37__Q0[0]=true
      break
      case 1
        doJ206_EtherCAT_Box_1__CPX_FB37__Q1[0]=true
      break
      case 2
        doJ206_EtherCAT_Box_1__CPX_FB37__Q2[0]=true
      break
      case 3
        doJ206_EtherCAT_Box_1__CPX_FB37__Q3[0]=true
      break
      case 4
        doJ206_EtherCAT_Box_1__CPX_FB37__Q4[0]=true
      break
      case 5
        doJ206_EtherCAT_Box_1__CPX_FB37__Q5[0]=true
      break
      case 6
        doJ206_EtherCAT_Box_1__CPX_FB37__Q6[0]=true
      break
      case 7
        doJ206_EtherCAT_Box_1__CPX_FB37__Q7[0]=true
      break
      case 8
        doJ206_EtherCAT_Box_1__CPX_FB37__Q8[0]=true
      break
      case 9
        doJ206_EtherCAT_Box_1__CPX_FB37__Q9[0]=true
      break
      case 10
        doJ206_EtherCAT_Box_1__CPX_FB37__Q10[0]=true
      break
      case 11
        doJ206_EtherCAT_Box_1__CPX_FB37__Q11[0]=true
      break
      case 12
        doJ206_EtherCAT_Box_1__CPX_FB37__Q12[0]=true
      break
      case 13
        doJ206_EtherCAT_Box_1__CPX_FB37__Q13[0]=true
      break
      case 14
        doJ206_EtherCAT_Box_1__CPX_FB37__Q14[0]=true
      break
      case 15
        doJ206_EtherCAT_Box_1__CPX_FB37__Q15[0]=true
      break
      case 16
        doJ206_EtherCAT_Box_1__CPX_FB37__Q16[0]=true
      break
      case 17
        doJ206_EtherCAT_Box_1__CPX_FB37__Q17[0]=true
      break
    endSwitch
  endIf

  // -- setup button colors for frontpage
  if statusValves[airexValve[0]] == 1 and statusValves[airexValve[1]] == 1  and statusValves[airexValve[2]] == 1 and  statusValves[airexValve[3]] == 1 and statusValves[airexValve[4]] == 1 and statusValves[airexValve[5]] == 1
    colorVacuumStatus1 = colorOn
  else
    colorVacuumStatus1 = colorOff
  endIf


end
